# EPICS autosave request: iocBoot/gmca_23i_ioc1/dbSave/RB_Rd_.req
%
% BURT Request File
%
% $(P)RB:Rd:  Robot dewar distances
%

file assy.req ASSY=$(P)RB:Rd

file mtr1.req MTR1=$(P)RB:mrx
file mtr1.req MTR1=$(P)RB:mry
file mtr1.req MTR1=$(P)RB:mrz

file drv1.req DRV1=$(P)RB:RX
file drv1.req DRV1=$(P)RB:RY
file drv1.req DRV1=$(P)RB:RZ
